// Mitsubishi GX Works2 project: G5CstCleaner   PLC: Q12H

PROGRAM MAIN
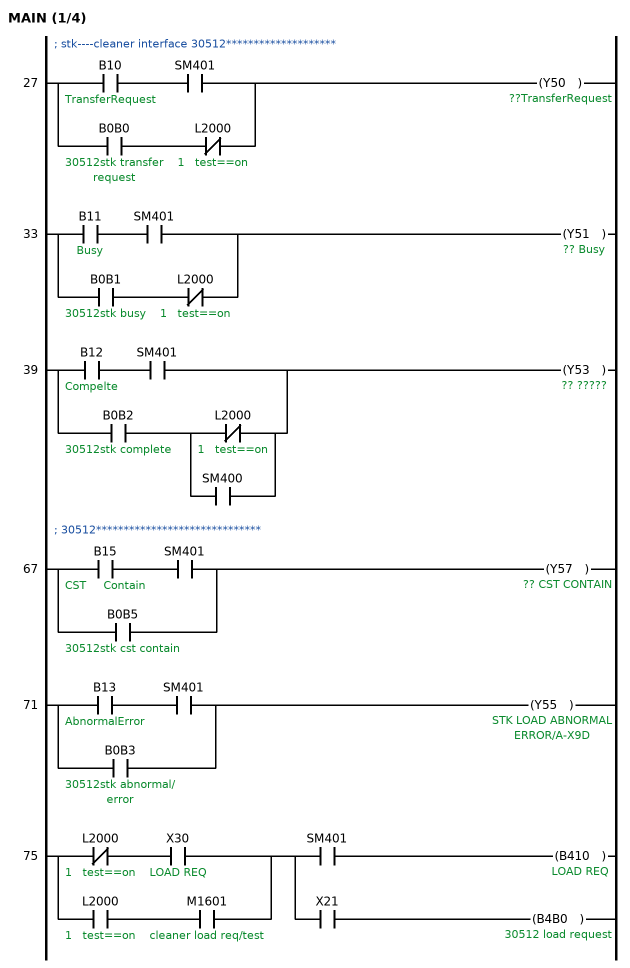
; stk----cleaner interface 30512********************
27    LD      B10  ; TransferRequest
      AND     SM401
      LD      B0B0  ; 30512stk transfer request
      ANI     L2000  ; 1   test==on
      ORB
      OUT     Y50  ; ??TransferRequest
33    LD      B11  ; Busy
      AND     SM401
      LD      B0B1  ; 30512stk busy
      ANI     L2000  ; 1   test==on
      ORB
      OUT     Y51  ; ?? Busy
39    LD      B12  ; Compelte
      AND     SM401
      LD      B0B2  ; 30512stk complete
      LDI     L2000  ; 1   test==on
      OR      SM400
      ANB
      ORB
      OUT     Y53  ; ?? ?????
; 30512******************************
67    LD      B15  ; CST     Contain
      AND     SM401
      OR      B0B5  ; 30512stk cst contain
      OUT     Y57  ; ?? CST CONTAIN
71    LD      B13  ; AbnormalError
      AND     SM401
      OR      B0B3  ; 30512stk abnormal/error
      OUT     Y55  ; STK LOAD ABNORMAL ERROR/A-X9D
75    LDI     L2000  ; 1   test==on
      AND     X30  ; LOAD REQ
      LD      L2000  ; 1   test==on
      AND     M1601  ; cleaner load req/test
      ORB
      MPS
      AND     SM401
      OUT     B410  ; LOAD REQ
      MPP
      AND     X21
      OUT     B4B0  ; 30512 load request
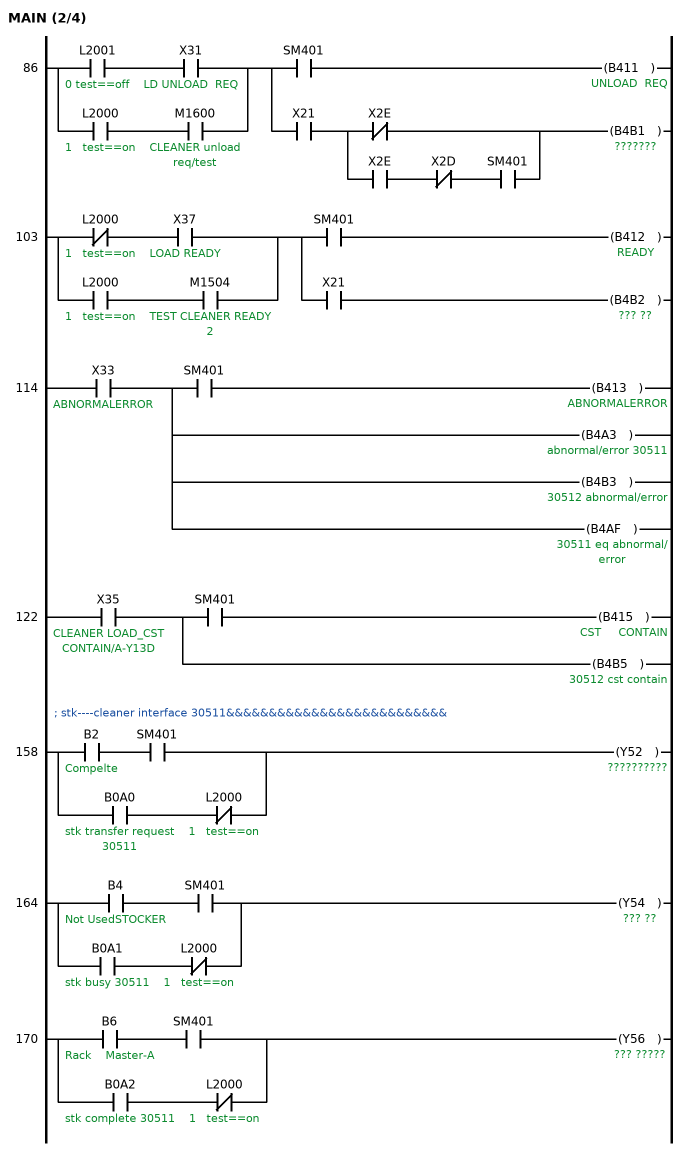
86    LD      L2001  ; 0 test==off
      AND     X31  ; LD UNLOAD  REQ
      LD      L2000  ; 1   test==on
      AND     M1600  ; CLEANER unload req/test
      ORB
      MPS
      AND     SM401
      OUT     B411  ; UNLOAD  REQ
      MPP
      AND     X21
      LDI     X2E
      LD      X2E
      ANI     X2D
      AND     SM401
      ORB
      ANB
      OUT     B4B1  ; ???????
103   LDI     L2000  ; 1   test==on
      AND     X37  ; LOAD READY
      LD      L2000  ; 1   test==on
      AND     M1504  ; TEST CLEANER READY 2
      ORB
      MPS
      AND     SM401
      OUT     B412  ; READY
      MPP
      AND     X21
      OUT     B4B2  ; ??? ??
114   LD      X33  ; ABNORMALERROR
      MPS
      AND     SM401
      OUT     B413  ; ABNORMALERROR
      MPP
      OUT     B4A3  ; abnormal/error 30511
      OUT     B4B3  ; 30512 abnormal/error
      OUT     B4AF  ; 30511 eq abnormal/error
122   LD      X35  ; CLEANER LOAD_CST CONTAIN/A-Y13D
      MPS
      AND     SM401
      OUT     B415  ; CST     CONTAIN
      MPP
      OUT     B4B5  ; 30512 cst contain
; stk----cleaner interface 30511&&&&&&&&&&&&&&&&&&&&&&&&&&
158   LD      B2  ; Compelte
      AND     SM401
      LD      B0A0  ; stk transfer request 30511
      ANI     L2000  ; 1   test==on
      ORB
      OUT     Y52  ; ??????????
164   LD      B4  ; Not UsedSTOCKER
      AND     SM401
      LD      B0A1  ; stk busy 30511
      ANI     L2000  ; 1   test==on
      ORB
      OUT     Y54  ; ??? ??
170   LD      B6  ; Rack    Master-A
      AND     SM401
      LD      B0A2  ; stk complete 30511
      ANI     L2000  ; 1   test==on
      ORB
      OUT     Y56  ; ??? ?????
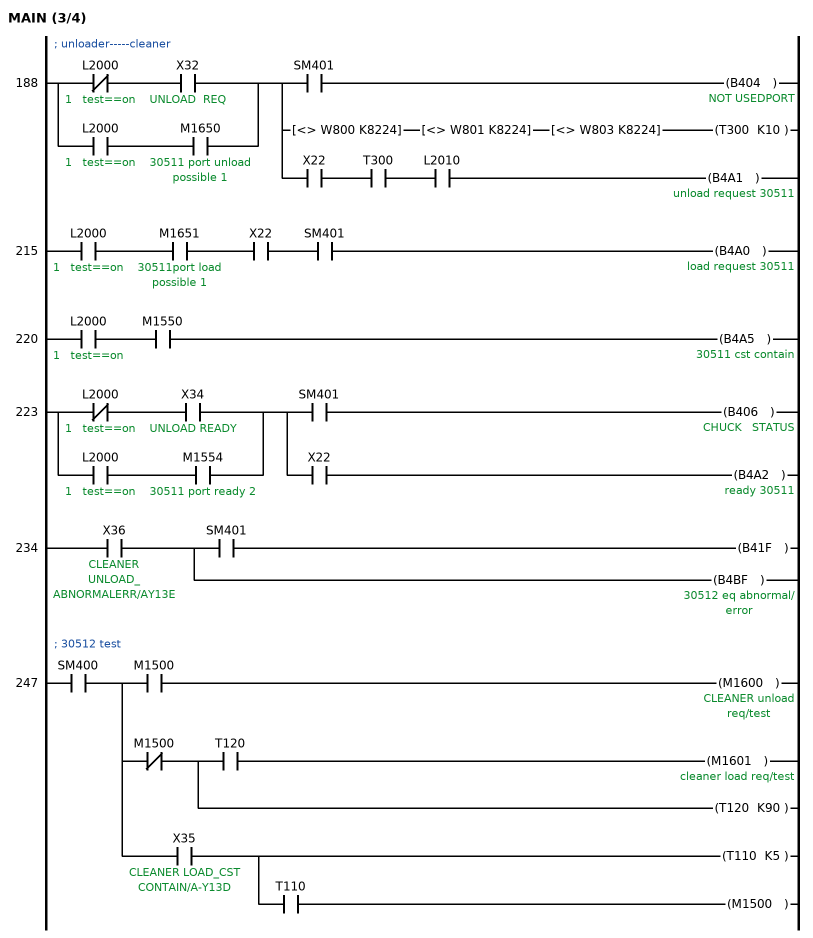
; unloader-----cleaner
188   LDI     L2000  ; 1   test==on
      AND     X32  ; UNLOAD  REQ
      LD      L2000  ; 1   test==on
      AND     M1650  ; 30511 port unload possible 1
      ORB
      MPS
      AND     SM401
      OUT     B404  ; NOT USEDPORT
      MRD
      AND<>   W800 K8224
      AND<>   W801 K8224
      AND<>   W803 K8224
      OUT     T300 K10
      MPP
      AND     X22
      AND     T300
      AND     L2010
      OUT     B4A1  ; unload request 30511
215   LD      L2000  ; 1   test==on
      AND     M1651  ; 30511port load possible 1
      AND     X22
      AND     SM401
      OUT     B4A0  ; load request 30511
220   LD      L2000  ; 1   test==on
      AND     M1550
      OUT     B4A5  ; 30511 cst contain
223   LDI     L2000  ; 1   test==on
      AND     X34  ; UNLOAD READY
      LD      L2000  ; 1   test==on
      AND     M1554  ; 30511 port ready 2
      ORB
      MPS
      AND     SM401
      OUT     B406  ; CHUCK   STATUS
      MPP
      AND     X22
      OUT     B4A2  ; ready 30511
234   LD      X36  ; CLEANER UNLOAD_ABNORMALERR/AY13E
      MPS
      AND     SM401
      OUT     B41F
      MPP
      OUT     B4BF  ; 30512 eq abnormal/error
; 30512 test
247   LD      SM400
      MPS
      AND     M1500
      OUT     M1600  ; CLEANER unload req/test
      MRD
      ANI     M1500
      MPS
      AND     T120
      OUT     M1601  ; cleaner load req/test
      MPP
      OUT     T120 K90
      MPP
      AND     X35  ; CLEANER LOAD_CST CONTAIN/A-Y13D
      OUT     T110 K5
      AND     T110
      OUT     M1500
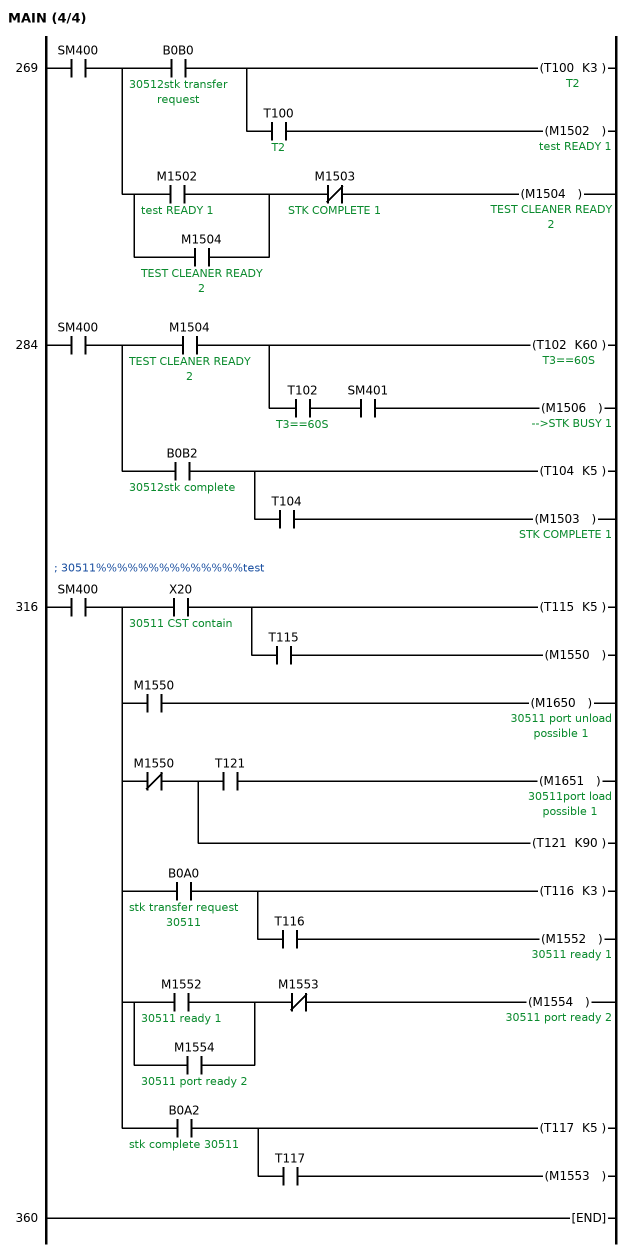
269   LD      SM400
      MPS
      AND     B0B0  ; 30512stk transfer request
      OUT     T100 K3  ; T2
      AND     T100  ; T2
      OUT     M1502  ; test READY 1
      MPP
      LD      M1502  ; test READY 1
      OR      M1504  ; TEST CLEANER READY 2
      ANB
      ANI     M1503  ; STK COMPLETE 1
      OUT     M1504  ; TEST CLEANER READY 2
284   LD      SM400
      MPS
      AND     M1504  ; TEST CLEANER READY 2
      OUT     T102 K60  ; T3==60S
      AND     T102  ; T3==60S
      AND     SM401
      OUT     M1506  ; -->STK BUSY 1
      MPP
      AND     B0B2  ; 30512stk complete
      OUT     T104 K5
      AND     T104
      OUT     M1503  ; STK COMPLETE 1
; 30511%%%%%%%%%%%%%%test
316   LD      SM400
      MPS
      AND     X20  ; 30511 CST contain
      OUT     T115 K5
      AND     T115
      OUT     M1550
      MRD
      AND     M1550
      OUT     M1650  ; 30511 port unload possible 1
      MRD
      ANI     M1550
      MPS
      AND     T121
      OUT     M1651  ; 30511port load possible 1
      MPP
      OUT     T121 K90
      MRD
      AND     B0A0  ; stk transfer request 30511
      OUT     T116 K3
      AND     T116
      OUT     M1552  ; 30511 ready 1
      MRD
      LD      M1552  ; 30511 ready 1
      OR      M1554  ; 30511 port ready 2
      ANB
      ANI     M1553
      OUT     M1554  ; 30511 port ready 2
      MPP
      AND     B0A2  ; stk complete 30511
      OUT     T117 K5
      AND     T117
      OUT     M1553
360   END
END_PROGRAM

PROGRAM ONE
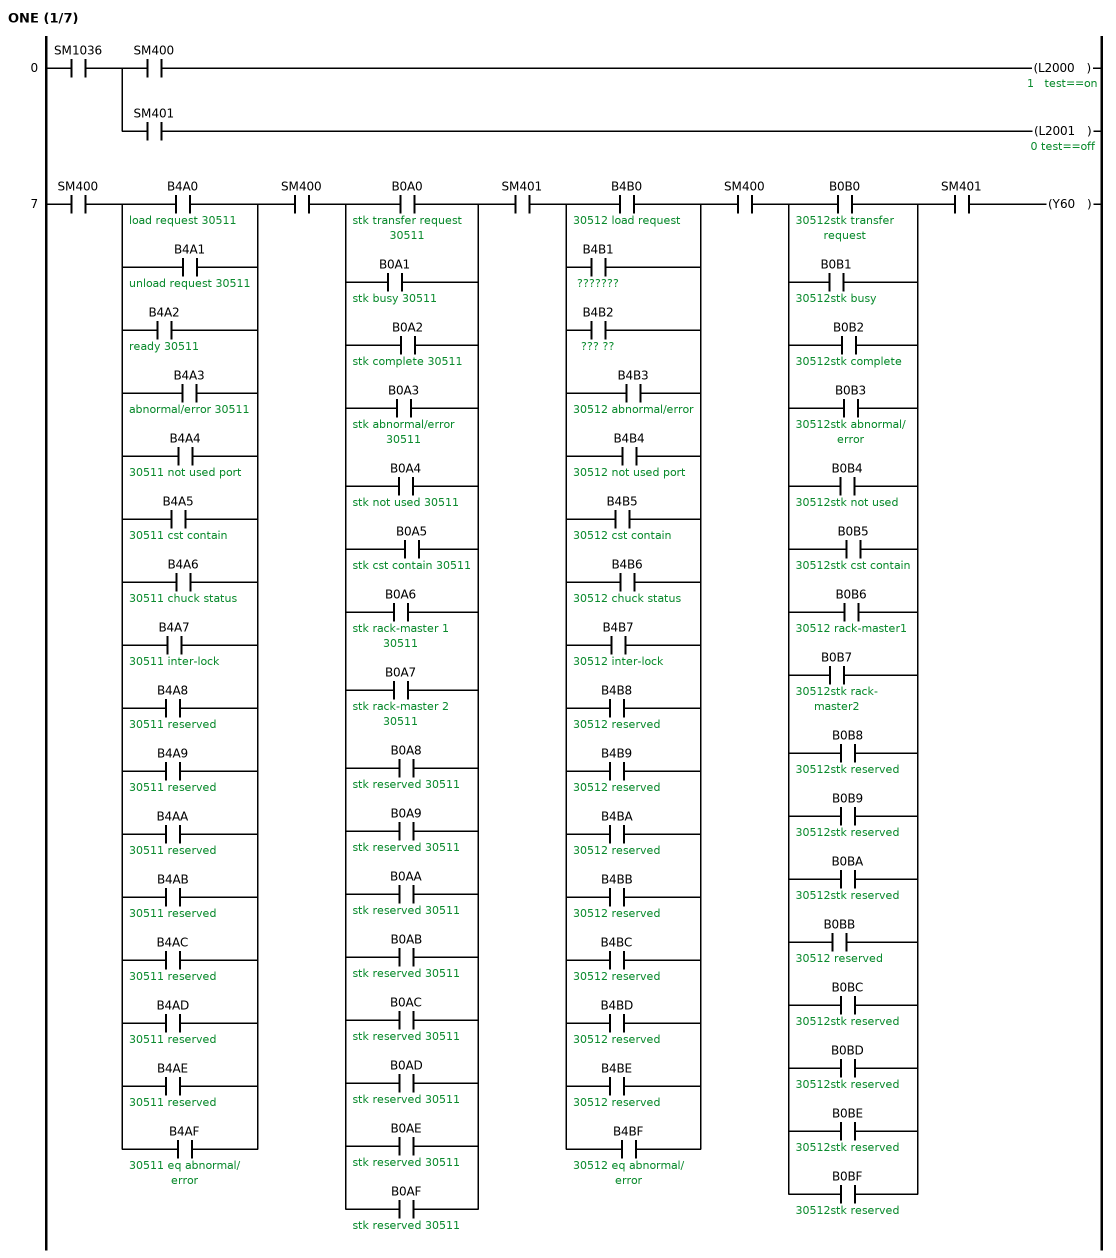
0     LD      SM1036
      MPS
      AND     SM400
      OUT     L2000  ; 1   test==on
      MPP
      AND     SM401
      OUT     L2001  ; 0 test==off
7     LD      SM400
      LD      B4A0  ; load request 30511
      OR      B4A1  ; unload request 30511
      OR      B4A2  ; ready 30511
      OR      B4A3  ; abnormal/error 30511
      OR      B4A4  ; 30511 not used port
      OR      B4A5  ; 30511 cst contain
      OR      B4A6  ; 30511 chuck status
      OR      B4A7  ; 30511 inter-lock
      OR      B4A8  ; 30511 reserved
      OR      B4A9  ; 30511 reserved
      OR      B4AA  ; 30511 reserved
      OR      B4AB  ; 30511 reserved
      OR      B4AC  ; 30511 reserved
      OR      B4AD  ; 30511 reserved
      OR      B4AE  ; 30511 reserved
      OR      B4AF  ; 30511 eq abnormal/error
      ANB
      AND     SM400
      LD      B0A0  ; stk transfer request 30511
      OR      B0A1  ; stk busy 30511
      OR      B0A2  ; stk complete 30511
      OR      B0A3  ; stk abnormal/error 30511
      OR      B0A4  ; stk not used 30511
      OR      B0A5  ; stk cst contain 30511
      OR      B0A6  ; stk rack-master 1 30511
      OR      B0A7  ; stk rack-master 2 30511
      OR      B0A8  ; stk reserved 30511
      OR      B0A9  ; stk reserved 30511
      OR      B0AA  ; stk reserved 30511
      OR      B0AB  ; stk reserved 30511
      OR      B0AC  ; stk reserved 30511
      OR      B0AD  ; stk reserved 30511
      OR      B0AE  ; stk reserved 30511
      OR      B0AF  ; stk reserved 30511
      ANB
      AND     SM401
      LD      B4B0  ; 30512 load request
      OR      B4B1  ; ???????
      OR      B4B2  ; ??? ??
      OR      B4B3  ; 30512 abnormal/error
      OR      B4B4  ; 30512 not used port
      OR      B4B5  ; 30512 cst contain
      OR      B4B6  ; 30512 chuck status
      OR      B4B7  ; 30512 inter-lock
      OR      B4B8  ; 30512 reserved
      OR      B4B9  ; 30512 reserved
      OR      B4BA  ; 30512 reserved
      OR      B4BB  ; 30512 reserved
      OR      B4BC  ; 30512 reserved
      OR      B4BD  ; 30512 reserved
      OR      B4BE  ; 30512 reserved
      OR      B4BF  ; 30512 eq abnormal/error
      ANB
      AND     SM400
      LD      B0B0  ; 30512stk transfer request
      OR      B0B1  ; 30512stk busy
      OR      B0B2  ; 30512stk complete
      OR      B0B3  ; 30512stk abnormal/error
      OR      B0B4  ; 30512stk not used
      OR      B0B5  ; 30512stk cst contain
      OR      B0B6  ; 30512 rack-master1
      OR      B0B7  ; 30512stk rack-master2
      OR      B0B8  ; 30512stk reserved
      OR      B0B9  ; 30512stk reserved
      OR      B0BA  ; 30512stk reserved
      OR      B0BB  ; 30512 reserved
      OR      B0BC  ; 30512stk reserved
      OR      B0BD  ; 30512stk reserved
      OR      B0BE  ; 30512stk reserved
      OR      B0BF  ; 30512stk reserved
      ANB
      AND     SM401
      OUT     Y60
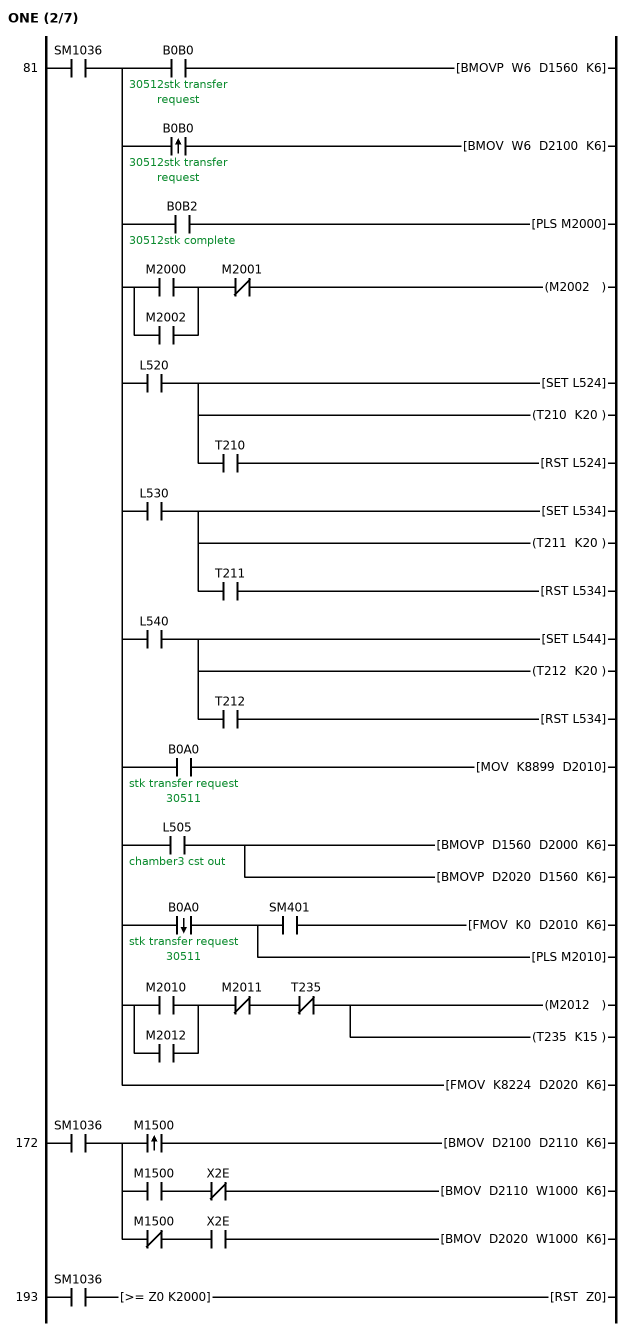
81    LD      SM1036
      MPS
      AND     B0B0  ; 30512stk transfer request
      BMOVP   W6 D1560 K6
      MRD
      ANDP    B0B0  ; 30512stk transfer request
      BMOV    W6 D2100 K6
      MRD
      AND     B0B2  ; 30512stk complete
      PLS     M2000
      MRD
      LD      M2000
      OR      M2002
      ANB
      ANI     M2001
      OUT     M2002
      MRD
      AND     L520
      SET     L524
      OUT     T210 K20
      AND     T210
      RST     L524
      MRD
      AND     L530
      SET     L534
      OUT     T211 K20
      AND     T211
      RST     L534
      MRD
      AND     L540
      SET     L544
      OUT     T212 K20
      AND     T212
      RST     L534
      MRD
      AND     B0A0  ; stk transfer request 30511
      MOV     K8899 D2010
      MRD
      AND     L505  ; chamber3 cst out
      BMOVP   D1560 D2000 K6
      BMOVP   D2020 D1560 K6
      MRD
      ANDF    B0A0  ; stk transfer request 30511
      MPS
      AND     SM401
      FMOV    K0 D2010 K6
      MPP
      PLS     M2010
      MRD
      LD      M2010
      OR      M2012
      ANB
      ANI     M2011
      ANI     T235
      OUT     M2012
      OUT     T235 K15
      MPP
      FMOV    K8224 D2020 K6
172   LD      SM1036
      MPS
      ANDP    M1500
      BMOV    D2100 D2110 K6
      MRD
      AND     M1500
      ANI     X2E
      BMOV    D2110 W1000 K6
      MPP
      ANI     M1500
      AND     X2E
      BMOV    D2020 W1000 K6
193   LD      SM1036
      AND>=   Z0 K2000
      RST     Z0
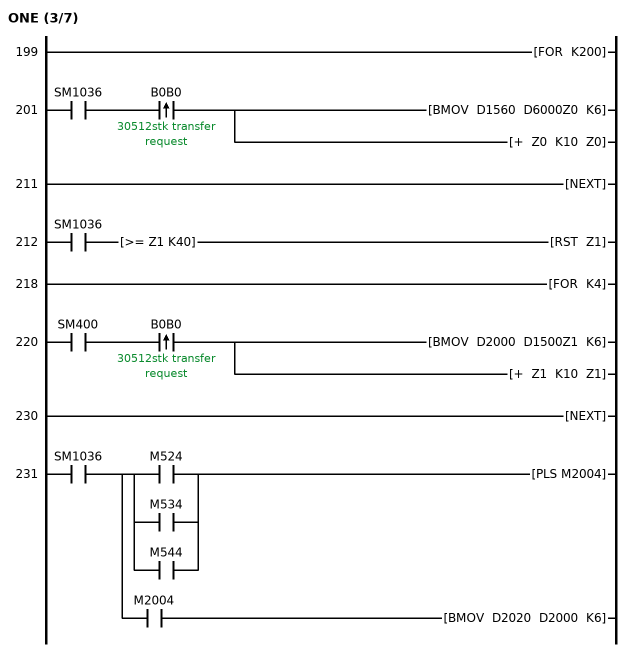
199   FOR     K200
201   LD      SM1036
      ANDP    B0B0  ; 30512stk transfer request
      BMOV    D1560 D6000Z0 K6
      +       Z0 K10 Z0
211   NEXT
212   LD      SM1036
      AND>=   Z1 K40
      RST     Z1
218   FOR     K4
220   LD      SM400
      ANDP    B0B0  ; 30512stk transfer request
      BMOV    D2000 D1500Z1 K6
      +       Z1 K10 Z1
230   NEXT
231   LD      SM1036
      MPS
      LD      M524
      OR      M534
      OR      M544
      ANB
      PLS     M2004
      MPP
      AND     M2004
      BMOV    D2020 D2000 K6
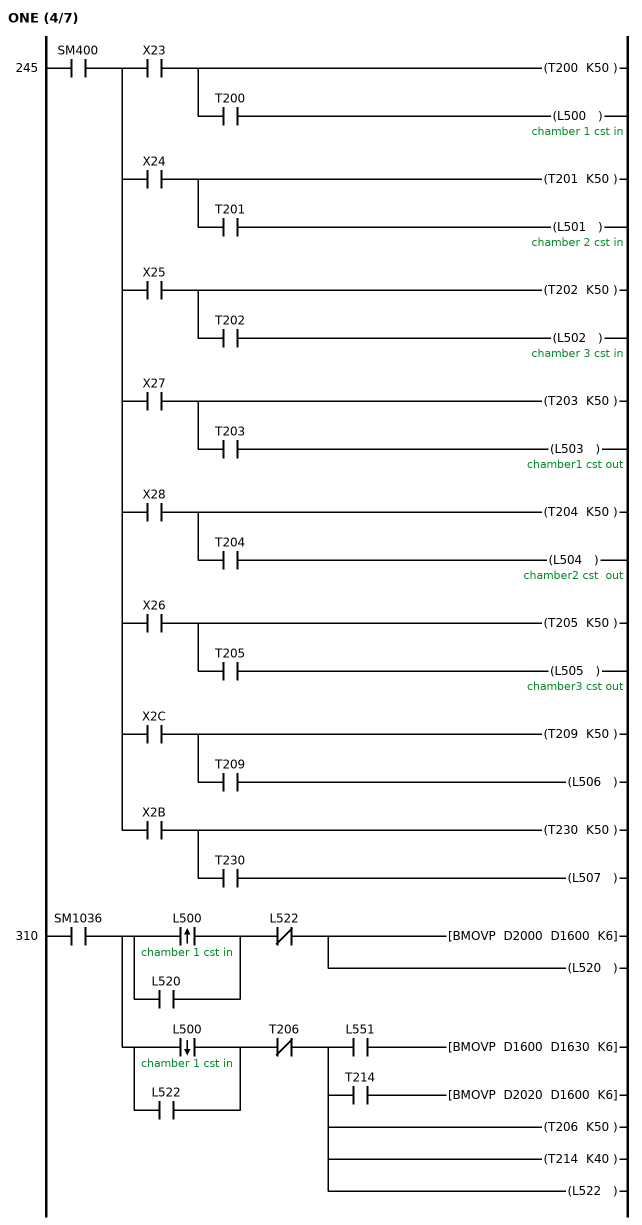
245   LD      SM400
      MPS
      AND     X23
      OUT     T200 K50
      AND     T200
      OUT     L500  ; chamber 1 cst in
      MRD
      AND     X24
      OUT     T201 K50
      AND     T201
      OUT     L501  ; chamber 2 cst in
      MRD
      AND     X25
      OUT     T202 K50
      AND     T202
      OUT     L502  ; chamber 3 cst in
      MRD
      AND     X27
      OUT     T203 K50
      AND     T203
      OUT     L503  ; chamber1 cst out
      MRD
      AND     X28
      OUT     T204 K50
      AND     T204
      OUT     L504  ; chamber2 cst  out
      MRD
      AND     X26
      OUT     T205 K50
      AND     T205
      OUT     L505  ; chamber3 cst out
      MRD
      AND     X2C
      OUT     T209 K50
      AND     T209
      OUT     L506
      MPP
      AND     X2B
      OUT     T230 K50
      AND     T230
      OUT     L507
310   LD      SM1036
      MPS
      LDP     L500  ; chamber 1 cst in
      OR      L520
      ANB
      ANI     L522
      BMOVP   D2000 D1600 K6
      OUT     L520
      MPP
      LDF     L500  ; chamber 1 cst in
      OR      L522
      ANB
      ANI     T206
      MPS
      AND     L551
      BMOVP   D1600 D1630 K6
      MRD
      AND     T214
      BMOVP   D2020 D1600 K6
      MPP
      OUT     T206 K50
      OUT     T214 K40
      OUT     L522
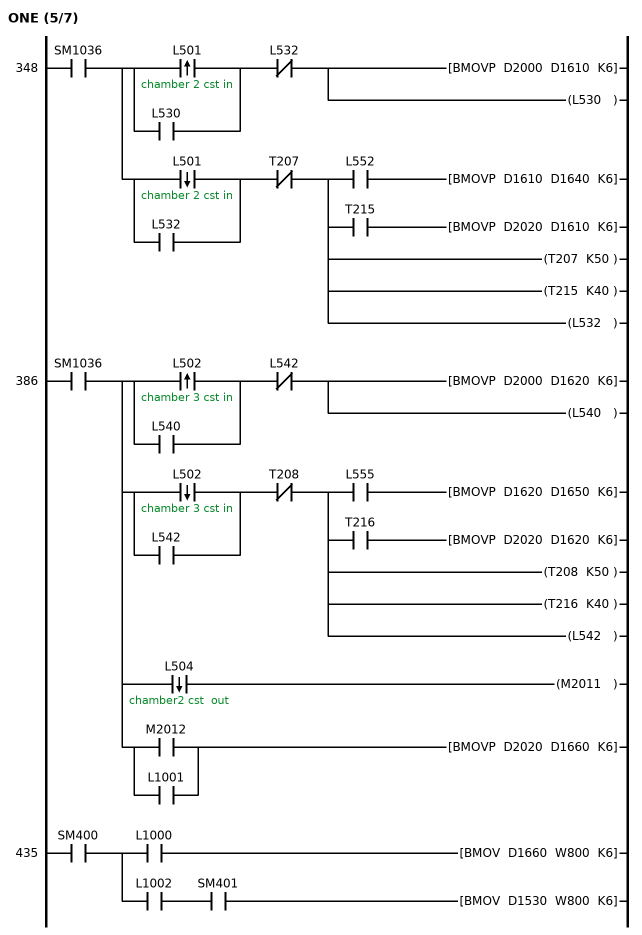
348   LD      SM1036
      MPS
      LDP     L501  ; chamber 2 cst in
      OR      L530
      ANB
      ANI     L532
      BMOVP   D2000 D1610 K6
      OUT     L530
      MPP
      LDF     L501  ; chamber 2 cst in
      OR      L532
      ANB
      ANI     T207
      MPS
      AND     L552
      BMOVP   D1610 D1640 K6
      MRD
      AND     T215
      BMOVP   D2020 D1610 K6
      MPP
      OUT     T207 K50
      OUT     T215 K40
      OUT     L532
386   LD      SM1036
      MPS
      LDP     L502  ; chamber 3 cst in
      OR      L540
      ANB
      ANI     L542
      BMOVP   D2000 D1620 K6
      OUT     L540
      MRD
      LDF     L502  ; chamber 3 cst in
      OR      L542
      ANB
      ANI     T208
      MPS
      AND     L555
      BMOVP   D1620 D1650 K6
      MRD
      AND     T216
      BMOVP   D2020 D1620 K6
      MPP
      OUT     T208 K50
      OUT     T216 K40
      OUT     L542
      MRD
      ANDF    L504  ; chamber2 cst  out
      OUT     M2011
      MPP
      LD      M2012
      OR      L1001
      ANB
      BMOVP   D2020 D1660 K6
435   LD      SM400
      MPS
      AND     L1000
      BMOV    D1660 W800 K6
      MPP
      AND     L1002
      AND     SM401
      BMOV    D1530 W800 K6
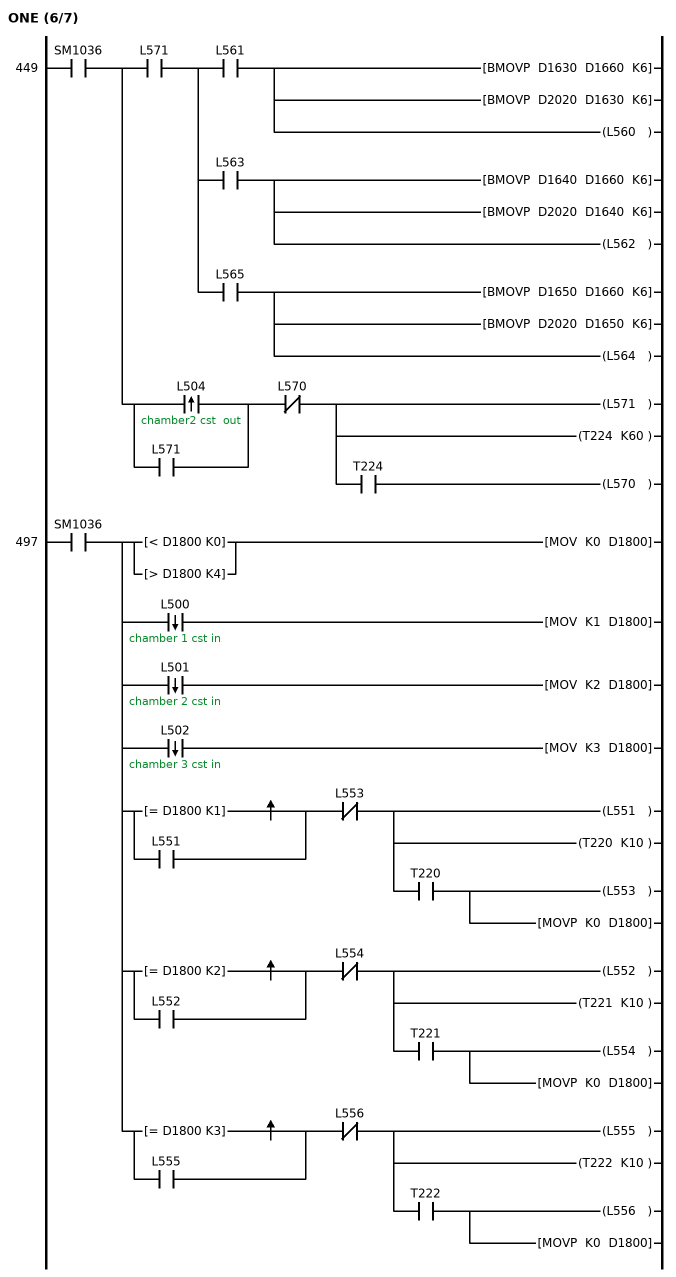
449   LD      SM1036
      MPS
      AND     L571
      MPS
      AND     L561
      BMOVP   D1630 D1660 K6
      BMOVP   D2020 D1630 K6
      OUT     L560
      MRD
      AND     L563
      BMOVP   D1640 D1660 K6
      BMOVP   D2020 D1640 K6
      OUT     L562
      MPP
      AND     L565
      BMOVP   D1650 D1660 K6
      BMOVP   D2020 D1650 K6
      OUT     L564
      MPP
      LDP     L504  ; chamber2 cst  out
      OR      L571
      ANB
      ANI     L570
      OUT     L571
      OUT     T224 K60
      AND     T224
      OUT     L570
497   LD      SM1036
      MPS
      LD<     D1800 K0
      OR>     D1800 K4
      ANB
      MOV     K0 D1800
      MRD
      ANDF    L500  ; chamber 1 cst in
      MOV     K1 D1800
      MRD
      ANDF    L501  ; chamber 2 cst in
      MOV     K2 D1800
      MRD
      ANDF    L502  ; chamber 3 cst in
      MOV     K3 D1800
      MRD
      LD=     D1800 K1
      MEP
      OR      L551
      ANB
      ANI     L553
      OUT     L551
      OUT     T220 K10
      AND     T220
      OUT     L553
      MOVP    K0 D1800
      MRD
      LD=     D1800 K2
      MEP
      OR      L552
      ANB
      ANI     L554
      OUT     L552
      OUT     T221 K10
      AND     T221
      OUT     L554
      MOVP    K0 D1800
      MPP
      LD=     D1800 K3
      MEP
      OR      L555
      ANB
      ANI     L556
      OUT     L555
      OUT     T222 K10
      AND     T222
      OUT     L556
      MOVP    K0 D1800
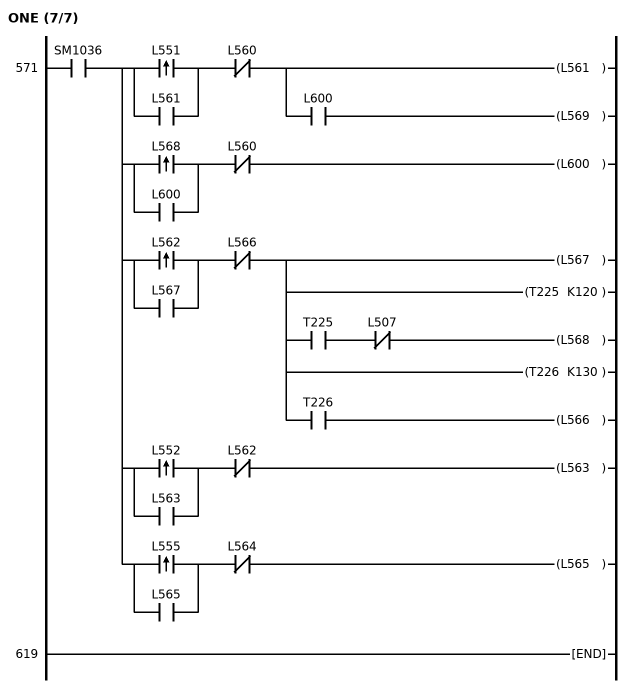
571   LD      SM1036
      MPS
      LDP     L551
      OR      L561
      ANB
      ANI     L560
      OUT     L561
      AND     L600
      OUT     L569
      MRD
      LDP     L568
      OR      L600
      ANB
      ANI     L560
      OUT     L600
      MRD
      LDP     L562
      OR      L567
      ANB
      ANI     L566
      OUT     L567
      OUT     T225 K120
      MPS
      AND     T225
      ANI     L507
      OUT     L568
      MPP
      OUT     T226 K130
      AND     T226
      OUT     L566
      MRD
      LDP     L552
      OR      L563
      ANB
      ANI     L562
      OUT     L563
      MPP
      LDP     L555
      OR      L565
      ANB
      ANI     L564
      OUT     L565
619   END
END_PROGRAM

PROGRAM ETHERNET
0     END
END_PROGRAM

// device comments not shown above
Y58  ; TransferRequest
Y59  ; Busy
Y5A  ; Compelte
Y5B  ; AbnormalError
Y5C  ; Not UsedSTOCKER
Y5D  ; CST     Contain
Y5E  ; Rack    Master-A
B0  ; TransferRequest
B1  ; Busy
B3  ; AbnormalError
B5  ; CST     Contain
B14  ; Not UsedSTOCKER
B16  ; Rack    Master-A
B400  ; LOAD REQ
B401  ; UNLOAD  REQ
B402  ; READY
B403  ; ABNORMALERROR
B405  ; CST     CONTAIN
B407  ; INTER    LOCK
B414  ; NOT USEDPORT
B416  ; CHUCK   STATUS
B417  ; INTER    LOCK
